// TIA Portal V19 export
FUNCTION_BLOCK "MainCabinetDiagReset"   // FB12, F_LAD
{ S7_Optimized_Access := 'TRUE' }
   VAR_INPUT
      RESET : Bool;
   END_VAR
BEGIN

REGION Network 1: 1=Acknowledgment for reintegration
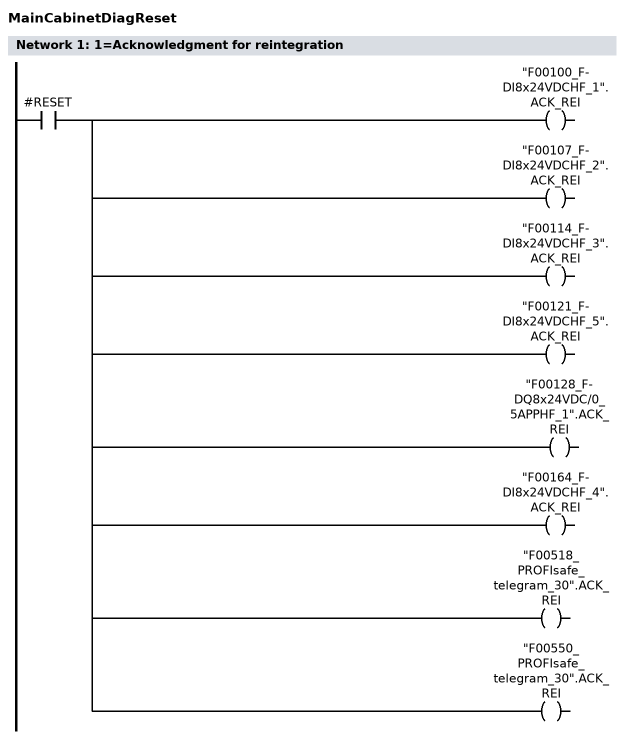
   RUNG wire#powerrail
      Contact( #RESET )
      wire#w1
      Coil( "F00100_F-DI8x24VDCHF_1".ACK_REI )
   END_RUNG
   RUNG wire#w1
      Coil( "F00107_F-DI8x24VDCHF_2".ACK_REI )
   END_RUNG
   RUNG wire#w1
      Coil( "F00114_F-DI8x24VDCHF_3".ACK_REI )
   END_RUNG
   RUNG wire#w1
      Coil( "F00121_F-DI8x24VDCHF_5".ACK_REI )
   END_RUNG
   RUNG wire#w1
      Coil( "F00128_F-DQ8x24VDC/0_5APPHF_1".ACK_REI )
   END_RUNG
   RUNG wire#w1
      Coil( "F00164_F-DI8x24VDCHF_4".ACK_REI )
   END_RUNG
   RUNG wire#w1
      Coil( "F00518_PROFIsafe_telegram_30".ACK_REI )
   END_RUNG
   RUNG wire#w1
      Coil( "F00550_PROFIsafe_telegram_30".ACK_REI )
   END_RUNG
   // the same network as SCL:
   "F00100_F-DI8x24VDCHF_1".ACK_REI := #RESET;
   "F00107_F-DI8x24VDCHF_2".ACK_REI := #RESET;
   "F00114_F-DI8x24VDCHF_3".ACK_REI := #RESET;
   "F00121_F-DI8x24VDCHF_5".ACK_REI := #RESET;
   "F00128_F-DQ8x24VDC/0_5APPHF_1".ACK_REI := #RESET;
   "F00164_F-DI8x24VDCHF_4".ACK_REI := #RESET;
   "F00518_PROFIsafe_telegram_30".ACK_REI := #RESET;
   "F00550_PROFIsafe_telegram_30".ACK_REI := #RESET;
END_REGION
END_FUNCTION_BLOCK
